(* Logix 5000 project; controller Sucrose_Main Emulate 5570 rev 20.12; software revision 20.01; part 5 of 30 *)
(* tags used below, declared in another part *)
   AI_E23_0 : REAL[8];   // Analog Input EN2T_FLX 192.168.1.23
   AI_E23_1 : REAL[8];   // Analog Input EN2T_FLX 192.168.1.23
   Alarm_ACK_Master_Timer : TIMER;
   CIPRemote : Area_Program;
   DI_E20_0 : ALIAS FOR FLX_E20:0:I;   // Discrete Input EN2T_FLX 192.168.1.20
   DI_E20_1 : ALIAS FOR FLX_E20:1:I;   // Discrete Input EN2T_FLX 192.168.1.20
   DO_E20_4 : ALIAS FOR FLX_E20:4:O;   // Discrete Output EN2T_FLX 192.168.1.20
   DO_E20_5 : ALIAS FOR FLX_E20:5:O;   // Discrete Output EN2T_FLX 192.168.1.20
   FV610501_AOI : QSI_Flow_Valve;   // FV-61-05-01-O CIP SUPPLY TO FILTRATION AND RING MAIN MIX PROOF VALVE OPEN
   FV620101_AOI : QSI_Flow_Valve;   // FV-62-01-01-O SUCROSE TANK #1 TO CIP RETURN PUMP MIX PROOF VALVE OPEN
   FV620201_AOI : QSI_Flow_Valve;   // FV-62-02-01-O SUCROSE TANK #2 TO CIP RETURN PUMP MIX PROOF VALVE OPEN
   Sucrose_MM_Enable : BOOL;
   SucroseCIP_PAUSED : BOOL;
   SucroseCIP_RINGMAIN_REMOTE : CIP_REMOTE;
   SucroseCIP_RUNNING : BOOL;
   SucroseCIP_SeatLift_Pulsing : BOOL;
   SucroseCIP_TK230101_REMOTE : CIP_REMOTE;
   SucroseCIP_TK230201_REMOTE : CIP_REMOTE;
   SucroseCIP_TK230301_REMOTE : CIP_REMOTE;
(* CIP_RemoteArea_AutoLogic, continued *)

ROUTINE CIP_TK230201_Remote   (* ladder *)
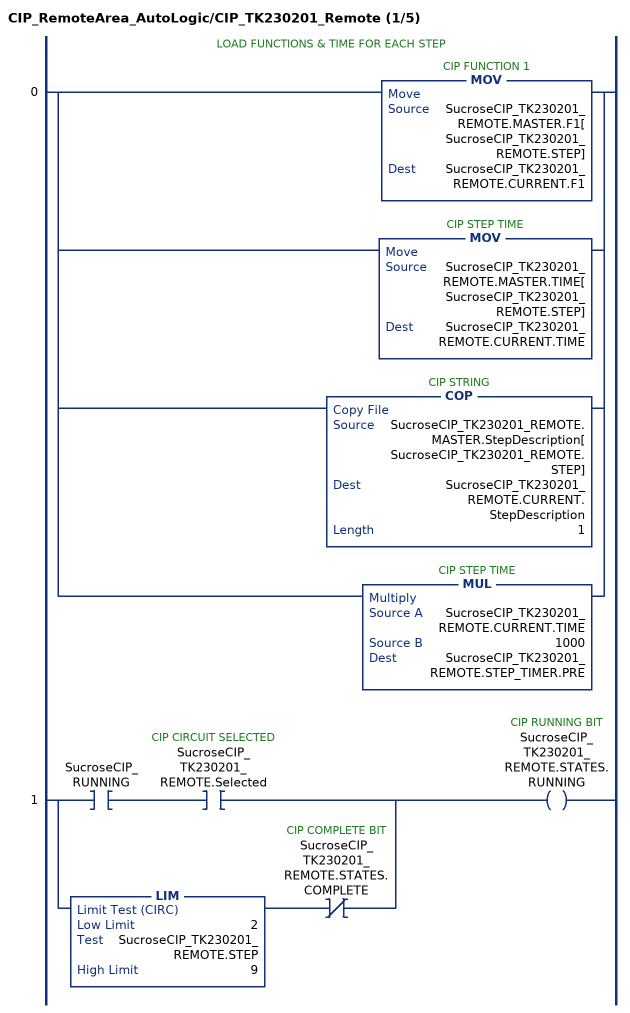
   // LOAD FUNCTIONS & TIME FOR EACH STEP
   0: [MOV(SucroseCIP_TK230201_REMOTE.MASTER.F1[SucroseCIP_TK230201_REMOTE.STEP],SucroseCIP_TK230201_REMOTE.CURRENT.F1) ,MOV(SucroseCIP_TK230201_REMOTE.MASTER.TIME[SucroseCIP_TK230201_REMOTE.STEP],SucroseCIP_TK230201_REMOTE.CURRENT.TIME) ,COP(SucroseCIP_TK230201_REMOTE.MASTER.StepDescription[SucroseCIP_TK230201_REMOTE.STEP],SucroseCIP_TK230201_REMOTE.CURRENT.StepDescription,1) ,MUL(SucroseCIP_TK230201_REMOTE.CURRENT.TIME,1000,SucroseCIP_TK230201_REMOTE.STEP_TIMER.PRE) ];
   1: [XIC(SucroseCIP_RUNNING) XIC(SucroseCIP_TK230201_REMOTE.Selected) ,LIM(2,SucroseCIP_TK230201_REMOTE.STEP,9) XIO(SucroseCIP_TK230201_REMOTE.STATES.COMPLETE) ]OTE(SucroseCIP_TK230201_REMOTE.STATES.RUNNING);
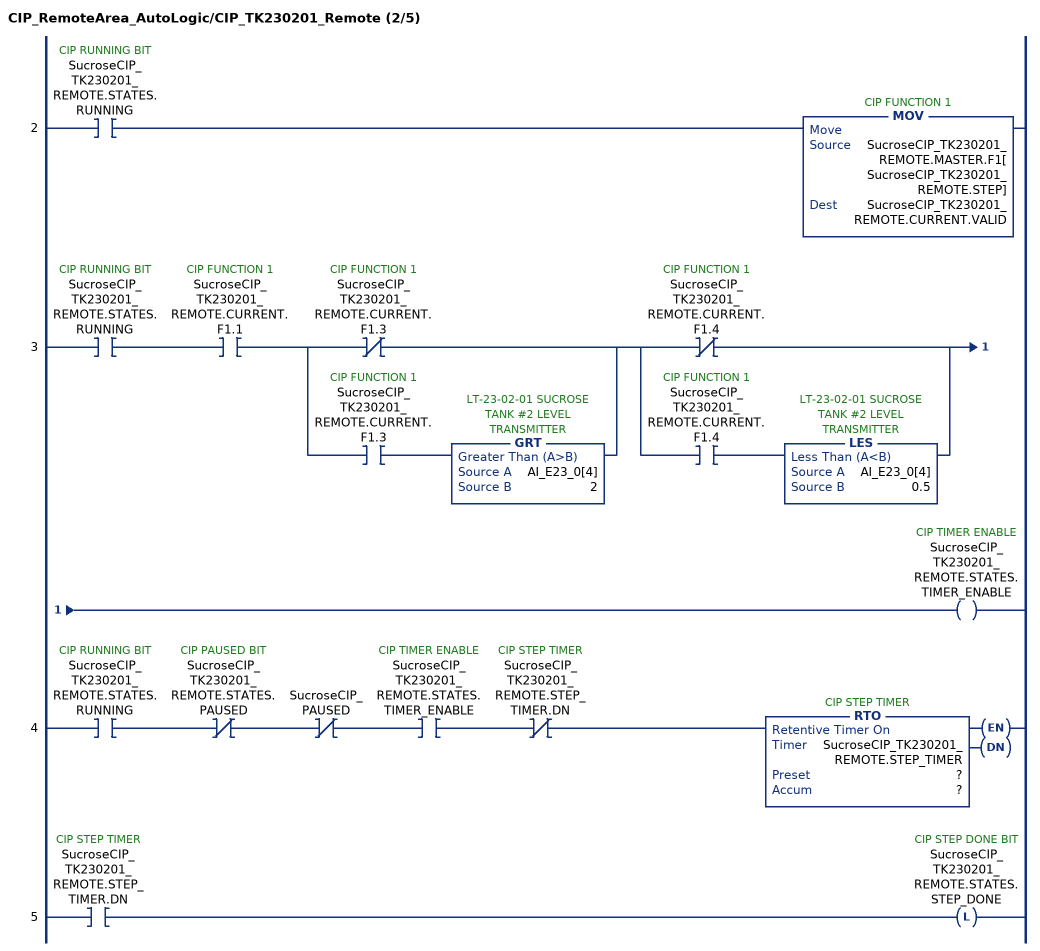
   2: XIC(SucroseCIP_TK230201_REMOTE.STATES.RUNNING)MOV(SucroseCIP_TK230201_REMOTE.MASTER.F1[SucroseCIP_TK230201_REMOTE.STEP],SucroseCIP_TK230201_REMOTE.CURRENT.VALID);
   3: XIC(SucroseCIP_TK230201_REMOTE.STATES.RUNNING)XIC(SucroseCIP_TK230201_REMOTE.CURRENT.F1.1)[XIO(SucroseCIP_TK230201_REMOTE.CURRENT.F1.3) ,XIC(SucroseCIP_TK230201_REMOTE.CURRENT.F1.3) GRT(AI_E23_0[4],2) ][XIO(SucroseCIP_TK230201_REMOTE.CURRENT.F1.4) ,XIC(SucroseCIP_TK230201_REMOTE.CURRENT.F1.4) LES(AI_E23_0[4],0.5) ]OTE(SucroseCIP_TK230201_REMOTE.STATES.TIMER_ENABLE);
   4: XIC(SucroseCIP_TK230201_REMOTE.STATES.RUNNING)XIO(SucroseCIP_TK230201_REMOTE.STATES.PAUSED)XIO(SucroseCIP_PAUSED)XIC(SucroseCIP_TK230201_REMOTE.STATES.TIMER_ENABLE)XIO(SucroseCIP_TK230201_REMOTE.STEP_TIMER.DN)RTO(SucroseCIP_TK230201_REMOTE.STEP_TIMER,?,?);
   5: XIC(SucroseCIP_TK230201_REMOTE.STEP_TIMER.DN)OTL(SucroseCIP_TK230201_REMOTE.STATES.STEP_DONE);
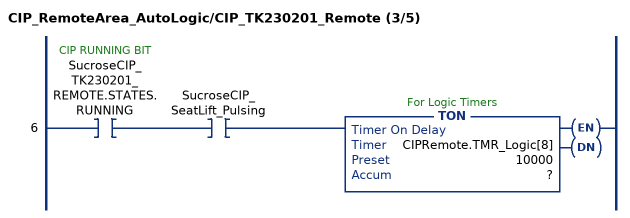
   6: XIC(SucroseCIP_TK230201_REMOTE.STATES.RUNNING)XIC(SucroseCIP_SeatLift_Pulsing)TON(CIPRemote.TMR_Logic[8],?,?);
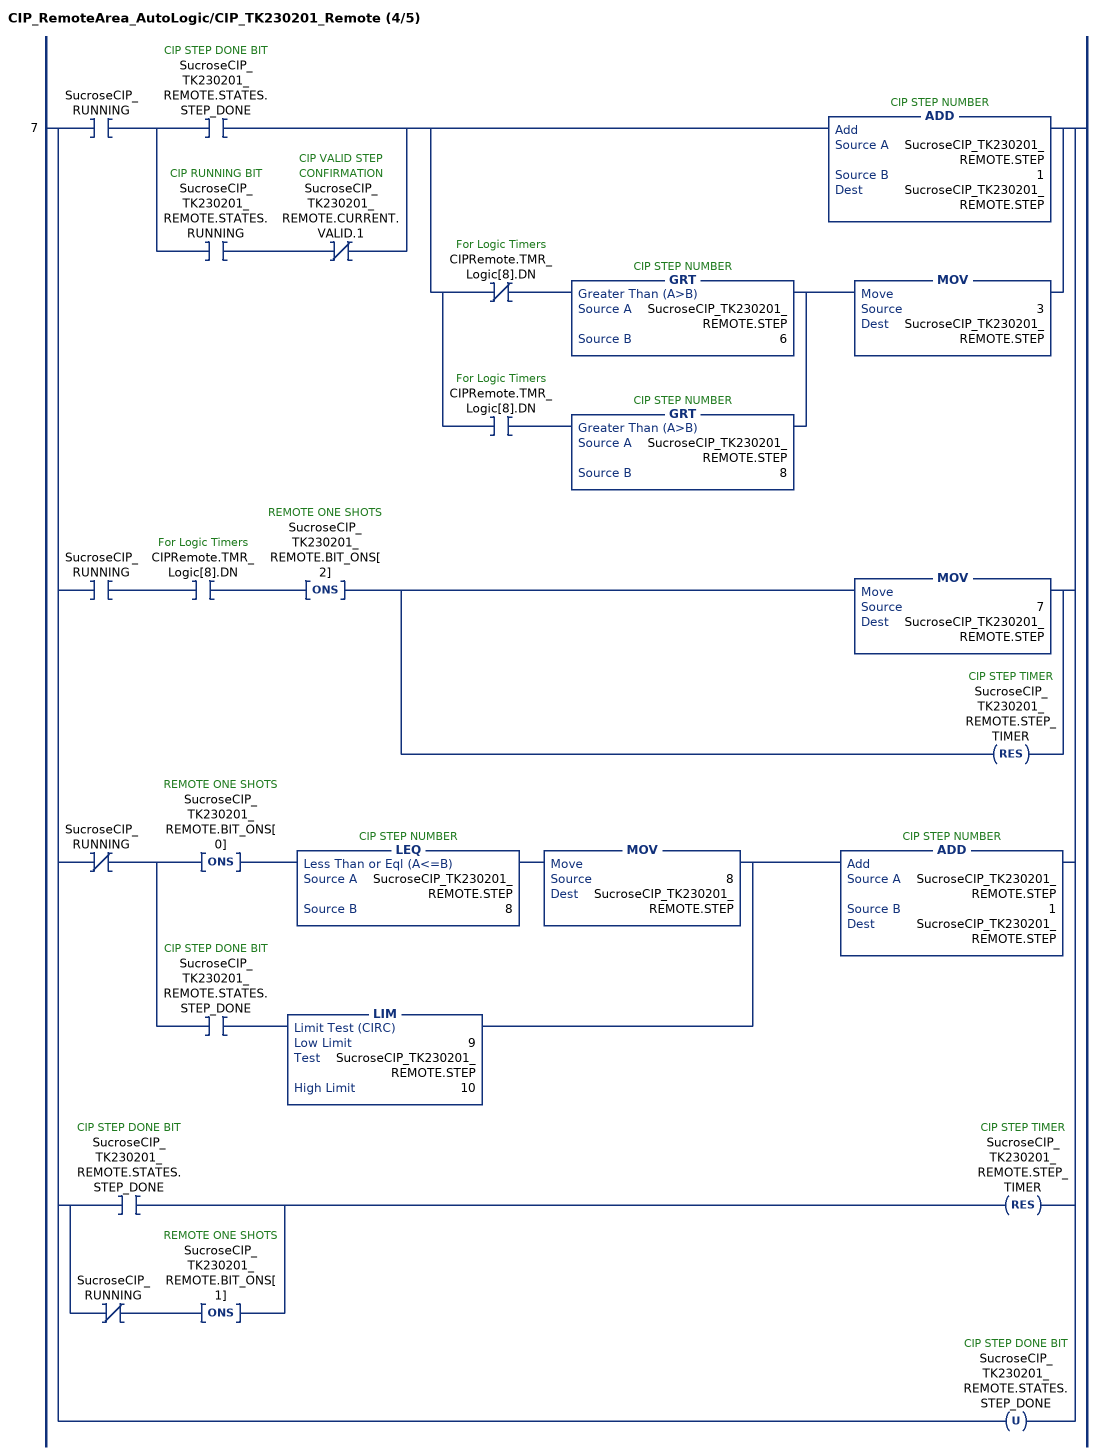
   7: [XIC(SucroseCIP_RUNNING) [XIC(SucroseCIP_TK230201_REMOTE.STATES.STEP_DONE) ,XIC(SucroseCIP_TK230201_REMOTE.STATES.RUNNING) XIO(SucroseCIP_TK230201_REMOTE.CURRENT.VALID.1) ] [ADD(SucroseCIP_TK230201_REMOTE.STEP,1,SucroseCIP_TK230201_REMOTE.STEP) ,[XIO(CIPRemote.TMR_Logic[8].DN) GRT(SucroseCIP_TK230201_REMOTE.STEP,6) ,XIC(CIPRemote.TMR_Logic[8].DN) GRT(SucroseCIP_TK230201_REMOTE.STEP,8) ] MOV(3,SucroseCIP_TK230201_REMOTE.STEP) ] ,XIC(SucroseCIP_RUNNING) XIC(CIPRemote.TMR_Logic[8].DN) ONS(SucroseCIP_TK230201_REMOTE.BIT_ONS[2]) [MOV(7,SucroseCIP_TK230201_REMOTE.STEP) ,RES(SucroseCIP_TK230201_REMOTE.STEP_TIMER) ] ,XIO(SucroseCIP_RUNNING) [ONS(SucroseCIP_TK230201_REMOTE.BIT_ONS[0]) LEQ(SucroseCIP_TK230201_REMOTE.STEP,8) MOV(8,SucroseCIP_TK230201_REMOTE.STEP) ,XIC(SucroseCIP_TK230201_REMOTE.STATES.STEP_DONE) LIM(9,SucroseCIP_TK230201_REMOTE.STEP,10) ] ADD(SucroseCIP_TK230201_REMOTE.STEP,1,SucroseCIP_TK230201_REMOTE.STEP) ,[XIC(SucroseCIP_TK230201_REMOTE.STATES.STEP_DONE) ,XIO(SucroseCIP_RUNNING) ONS(SucroseCIP_TK230201_REMOTE.BIT_ONS[1]) ] RES(SucroseCIP_TK230201_REMOTE.STEP_TIMER) ,OTU(SucroseCIP_TK230201_REMOTE.STATES.STEP_DONE) ];
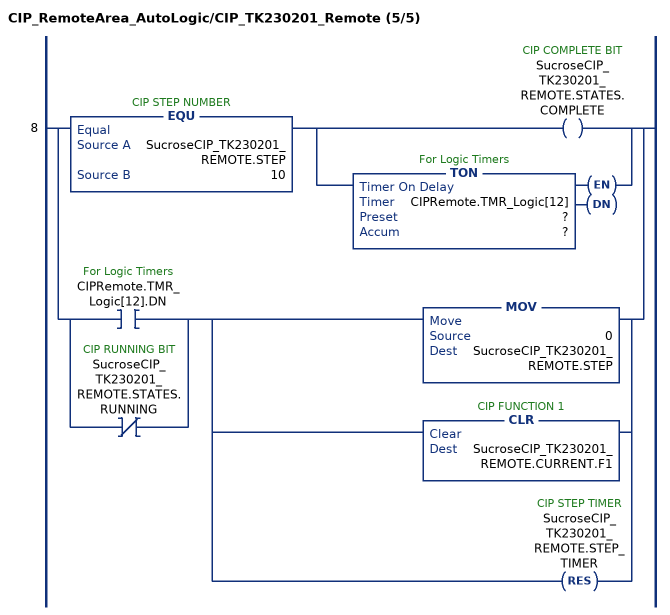
   8: [EQU(SucroseCIP_TK230201_REMOTE.STEP,10) [OTE(SucroseCIP_TK230201_REMOTE.STATES.COMPLETE) ,TON(CIPRemote.TMR_Logic[12],?,?) ] ,[XIC(CIPRemote.TMR_Logic[12].DN) ,XIO(SucroseCIP_TK230201_REMOTE.STATES.RUNNING) ] [MOV(0,SucroseCIP_TK230201_REMOTE.STEP) ,CLR(SucroseCIP_TK230201_REMOTE.CURRENT.F1) ,RES(SucroseCIP_TK230201_REMOTE.STEP_TIMER) ] ];
END_ROUTINE

ROUTINE CIP_TK230301_Remote   (* ladder *)
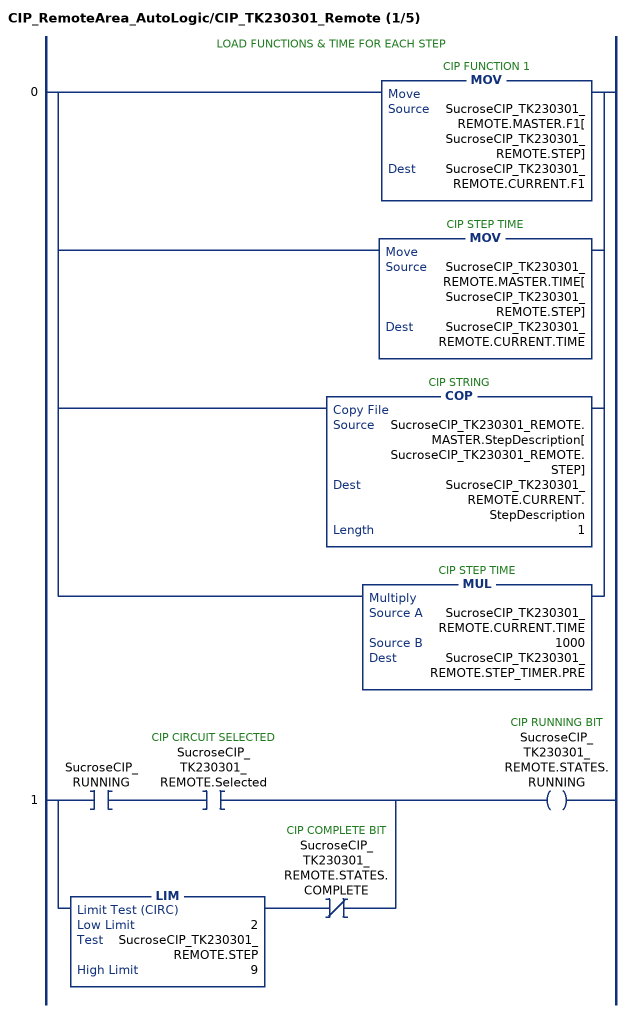
   // LOAD FUNCTIONS & TIME FOR EACH STEP
   0: [MOV(SucroseCIP_TK230301_REMOTE.MASTER.F1[SucroseCIP_TK230301_REMOTE.STEP],SucroseCIP_TK230301_REMOTE.CURRENT.F1) ,MOV(SucroseCIP_TK230301_REMOTE.MASTER.TIME[SucroseCIP_TK230301_REMOTE.STEP],SucroseCIP_TK230301_REMOTE.CURRENT.TIME) ,COP(SucroseCIP_TK230301_REMOTE.MASTER.StepDescription[SucroseCIP_TK230301_REMOTE.STEP],SucroseCIP_TK230301_REMOTE.CURRENT.StepDescription,1) ,MUL(SucroseCIP_TK230301_REMOTE.CURRENT.TIME,1000,SucroseCIP_TK230301_REMOTE.STEP_TIMER.PRE) ];
   1: [XIC(SucroseCIP_RUNNING) XIC(SucroseCIP_TK230301_REMOTE.Selected) ,LIM(2,SucroseCIP_TK230301_REMOTE.STEP,9) XIO(SucroseCIP_TK230301_REMOTE.STATES.COMPLETE) ]OTE(SucroseCIP_TK230301_REMOTE.STATES.RUNNING);
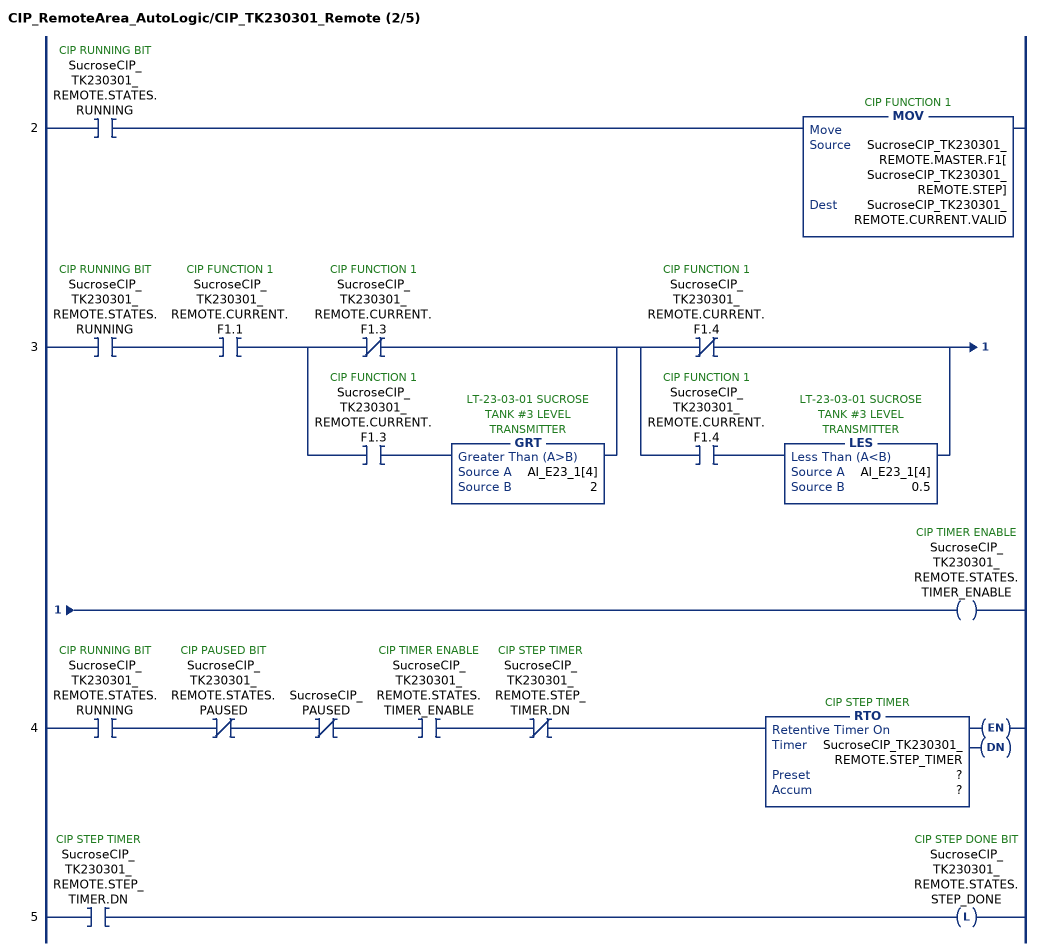
   2: XIC(SucroseCIP_TK230301_REMOTE.STATES.RUNNING)MOV(SucroseCIP_TK230301_REMOTE.MASTER.F1[SucroseCIP_TK230301_REMOTE.STEP],SucroseCIP_TK230301_REMOTE.CURRENT.VALID);
   3: XIC(SucroseCIP_TK230301_REMOTE.STATES.RUNNING)XIC(SucroseCIP_TK230301_REMOTE.CURRENT.F1.1)[XIO(SucroseCIP_TK230301_REMOTE.CURRENT.F1.3) ,XIC(SucroseCIP_TK230301_REMOTE.CURRENT.F1.3) GRT(AI_E23_1[4],2) ][XIO(SucroseCIP_TK230301_REMOTE.CURRENT.F1.4) ,XIC(SucroseCIP_TK230301_REMOTE.CURRENT.F1.4) LES(AI_E23_1[4],0.5) ]OTE(SucroseCIP_TK230301_REMOTE.STATES.TIMER_ENABLE);
   4: XIC(SucroseCIP_TK230301_REMOTE.STATES.RUNNING)XIO(SucroseCIP_TK230301_REMOTE.STATES.PAUSED)XIO(SucroseCIP_PAUSED)XIC(SucroseCIP_TK230301_REMOTE.STATES.TIMER_ENABLE)XIO(SucroseCIP_TK230301_REMOTE.STEP_TIMER.DN)RTO(SucroseCIP_TK230301_REMOTE.STEP_TIMER,?,?);
   5: XIC(SucroseCIP_TK230301_REMOTE.STEP_TIMER.DN)OTL(SucroseCIP_TK230301_REMOTE.STATES.STEP_DONE);
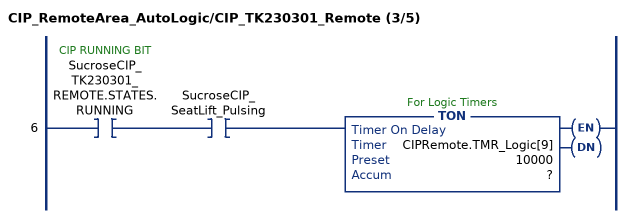
   6: XIC(SucroseCIP_TK230301_REMOTE.STATES.RUNNING)XIC(SucroseCIP_SeatLift_Pulsing)TON(CIPRemote.TMR_Logic[9],?,?);
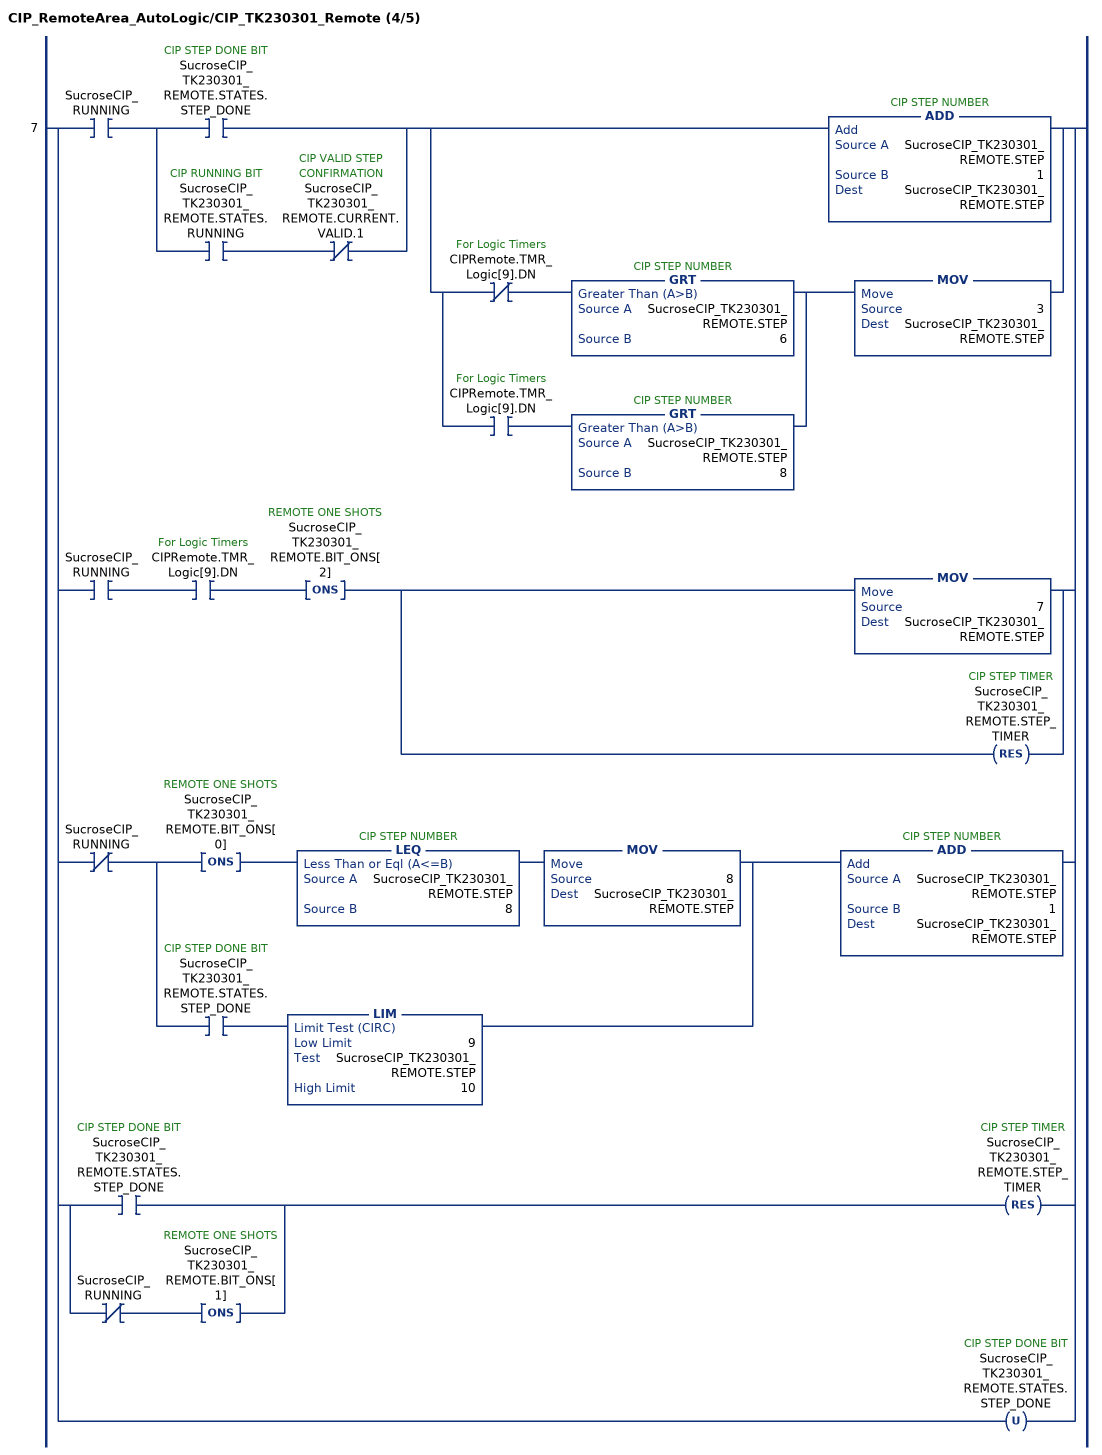
   7: [XIC(SucroseCIP_RUNNING) [XIC(SucroseCIP_TK230301_REMOTE.STATES.STEP_DONE) ,XIC(SucroseCIP_TK230301_REMOTE.STATES.RUNNING) XIO(SucroseCIP_TK230301_REMOTE.CURRENT.VALID.1) ] [ADD(SucroseCIP_TK230301_REMOTE.STEP,1,SucroseCIP_TK230301_REMOTE.STEP) ,[XIO(CIPRemote.TMR_Logic[9].DN) GRT(SucroseCIP_TK230301_REMOTE.STEP,6) ,XIC(CIPRemote.TMR_Logic[9].DN) GRT(SucroseCIP_TK230301_REMOTE.STEP,8) ] MOV(3,SucroseCIP_TK230301_REMOTE.STEP) ] ,XIC(SucroseCIP_RUNNING) XIC(CIPRemote.TMR_Logic[9].DN) ONS(SucroseCIP_TK230301_REMOTE.BIT_ONS[2]) [MOV(7,SucroseCIP_TK230301_REMOTE.STEP) ,RES(SucroseCIP_TK230301_REMOTE.STEP_TIMER) ] ,XIO(SucroseCIP_RUNNING) [ONS(SucroseCIP_TK230301_REMOTE.BIT_ONS[0]) LEQ(SucroseCIP_TK230301_REMOTE.STEP,8) MOV(8,SucroseCIP_TK230301_REMOTE.STEP) ,XIC(SucroseCIP_TK230301_REMOTE.STATES.STEP_DONE) LIM(9,SucroseCIP_TK230301_REMOTE.STEP,10) ] ADD(SucroseCIP_TK230301_REMOTE.STEP,1,SucroseCIP_TK230301_REMOTE.STEP) ,[XIC(SucroseCIP_TK230301_REMOTE.STATES.STEP_DONE) ,XIO(SucroseCIP_RUNNING) ONS(SucroseCIP_TK230301_REMOTE.BIT_ONS[1]) ] RES(SucroseCIP_TK230301_REMOTE.STEP_TIMER) ,OTU(SucroseCIP_TK230301_REMOTE.STATES.STEP_DONE) ];
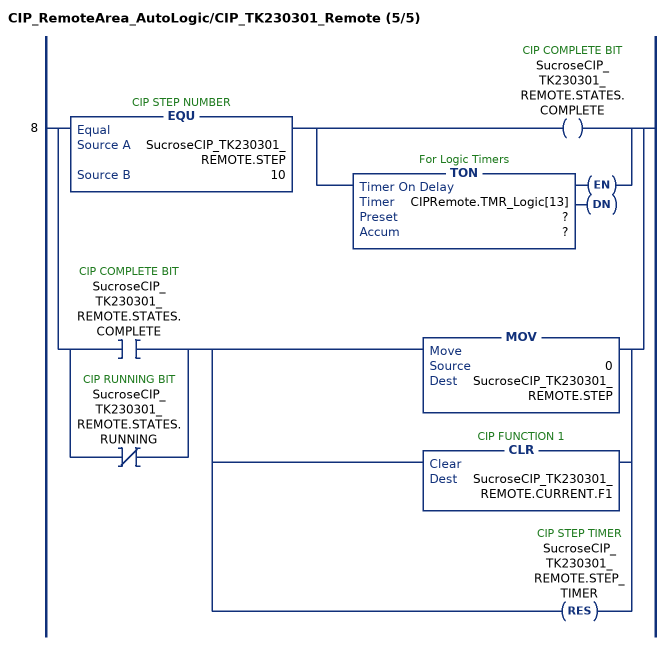
   8: [EQU(SucroseCIP_TK230301_REMOTE.STEP,10) [OTE(SucroseCIP_TK230301_REMOTE.STATES.COMPLETE) ,TON(CIPRemote.TMR_Logic[13],?,?) ] ,[XIC(SucroseCIP_TK230301_REMOTE.STATES.COMPLETE) ,XIO(SucroseCIP_TK230301_REMOTE.STATES.RUNNING) ] [MOV(0,SucroseCIP_TK230301_REMOTE.STEP) ,CLR(SucroseCIP_TK230301_REMOTE.CURRENT.F1) ,RES(SucroseCIP_TK230301_REMOTE.STEP_TIMER) ] ];
END_ROUTINE

ROUTINE MainRoutine   (* ladder *)
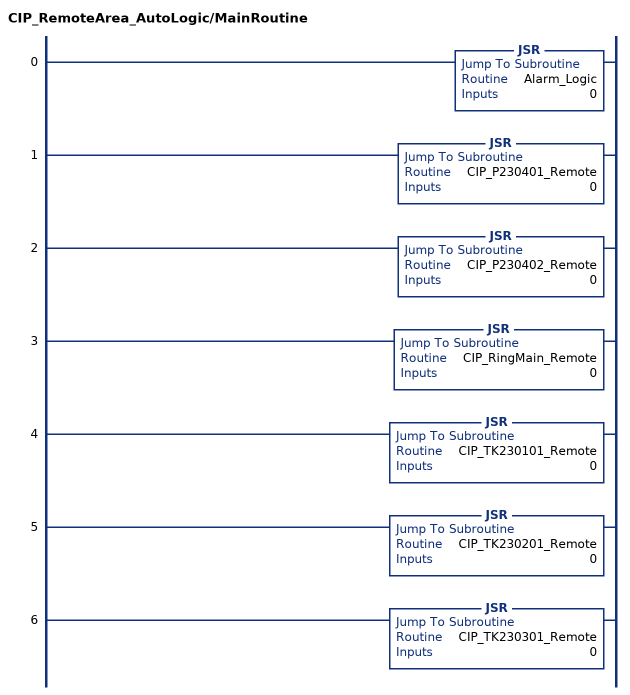
   0: JSR(Alarm_Logic,0);
   1: JSR(CIP_P230401_Remote,0);
   2: JSR(CIP_P230402_Remote,0);
   3: JSR(CIP_RingMain_Remote,0);
   4: JSR(CIP_TK230101_Remote,0);
   5: JSR(CIP_TK230201_Remote,0);
   6: JSR(CIP_TK230301_Remote,0);
END_ROUTINE
END_PROGRAM

PROGRAM CIP_RemoteArea_EN2T_IO_Discrete_DO_E20_4   (* main routine MainRoutine *)

ROUTINE _00_FV610501   (* ladder *)
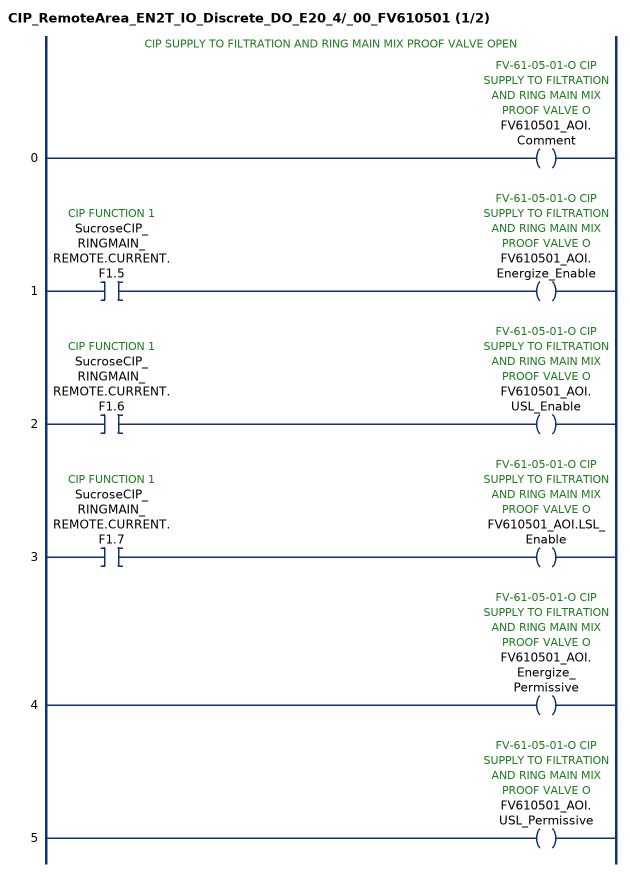
   // CIP SUPPLY TO FILTRATION AND RING MAIN MIX PROOF VALVE OPEN
   0: OTE(FV610501_AOI.Comment);
   1: XIC(SucroseCIP_RINGMAIN_REMOTE.CURRENT.F1.5)OTE(FV610501_AOI.Energize_Enable);
   2: XIC(SucroseCIP_RINGMAIN_REMOTE.CURRENT.F1.6)OTE(FV610501_AOI.USL_Enable);
   3: XIC(SucroseCIP_RINGMAIN_REMOTE.CURRENT.F1.7)OTE(FV610501_AOI.LSL_Enable);
   4: OTE(FV610501_AOI.Energize_Permissive);
   5: OTE(FV610501_AOI.USL_Permissive);
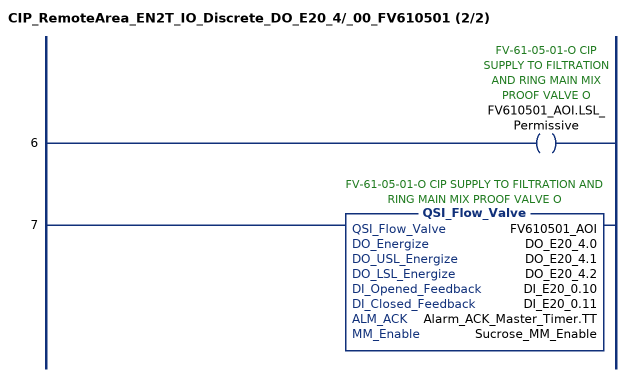
   6: OTE(FV610501_AOI.LSL_Permissive);
   7: QSI_Flow_Valve(FV610501_AOI,DO_E20_4.0,DO_E20_4.1,DO_E20_4.2,DI_E20_0.10,DI_E20_0.11,Alarm_ACK_Master_Timer.TT,Sucrose_MM_Enable);
END_ROUTINE

ROUTINE _12_FV620101   (* ladder *)
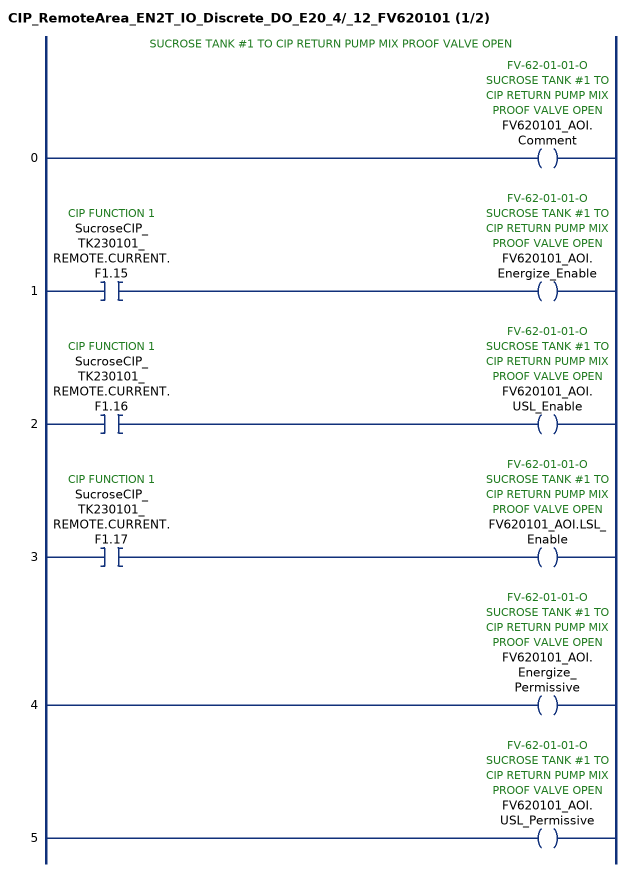
   // SUCROSE TANK #1 TO CIP RETURN PUMP MIX PROOF VALVE OPEN
   0: OTE(FV620101_AOI.Comment);
   1: XIC(SucroseCIP_TK230101_REMOTE.CURRENT.F1.15)OTE(FV620101_AOI.Energize_Enable);
   2: XIC(SucroseCIP_TK230101_REMOTE.CURRENT.F1.16)OTE(FV620101_AOI.USL_Enable);
   3: XIC(SucroseCIP_TK230101_REMOTE.CURRENT.F1.17)OTE(FV620101_AOI.LSL_Enable);
   4: OTE(FV620101_AOI.Energize_Permissive);
   5: OTE(FV620101_AOI.USL_Permissive);
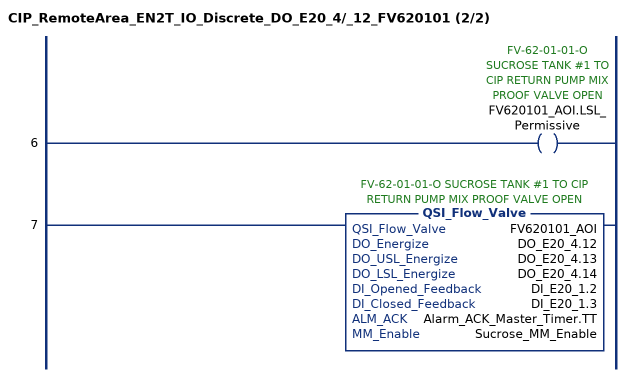
   6: OTE(FV620101_AOI.LSL_Permissive);
   7: QSI_Flow_Valve(FV620101_AOI,DO_E20_4.12,DO_E20_4.13,DO_E20_4.14,DI_E20_1.2,DI_E20_1.3,Alarm_ACK_Master_Timer.TT,Sucrose_MM_Enable);
END_ROUTINE

ROUTINE MainRoutine   (* ladder *)
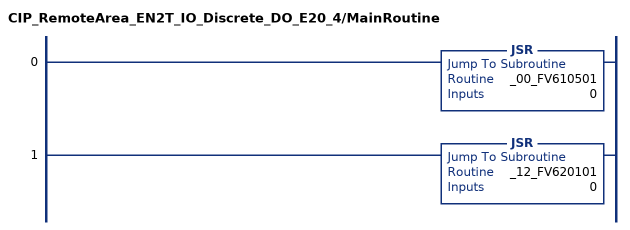
   0: JSR(_00_FV610501,0);
   1: JSR(_12_FV620101,0);
END_ROUTINE
END_PROGRAM

PROGRAM CIP_RemoteArea_EN2T_IO_Discrete_DO_E20_5   (* main routine MainRoutine *)

ROUTINE _00_FV620201   (* ladder *)
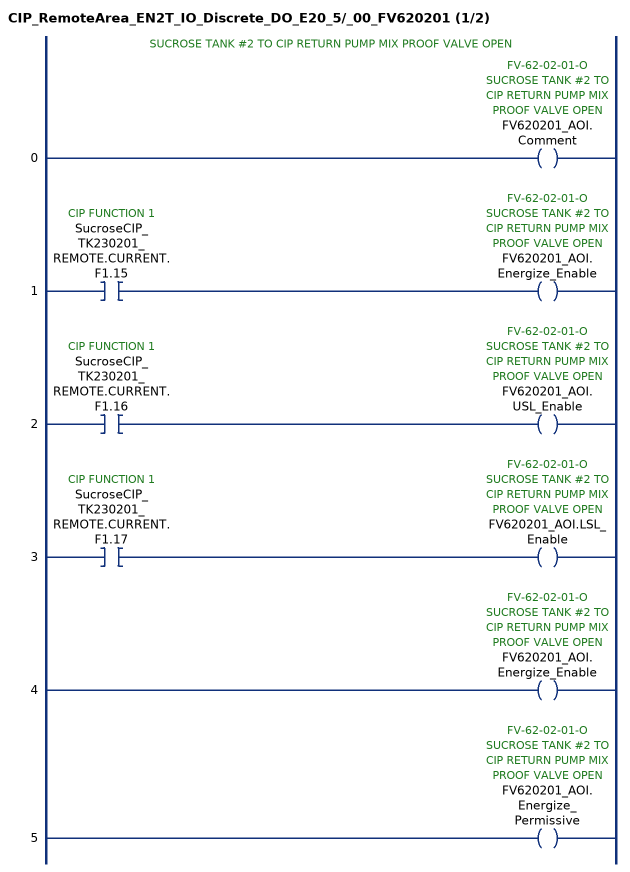
   // SUCROSE TANK #2 TO CIP RETURN PUMP MIX PROOF VALVE OPEN
   0: OTE(FV620201_AOI.Comment);
   1: XIC(SucroseCIP_TK230201_REMOTE.CURRENT.F1.15)OTE(FV620201_AOI.Energize_Enable);
   2: XIC(SucroseCIP_TK230201_REMOTE.CURRENT.F1.16)OTE(FV620201_AOI.USL_Enable);
   3: XIC(SucroseCIP_TK230201_REMOTE.CURRENT.F1.17)OTE(FV620201_AOI.LSL_Enable);
   4: OTE(FV620201_AOI.Energize_Enable);
   5: OTE(FV620201_AOI.Energize_Permissive);
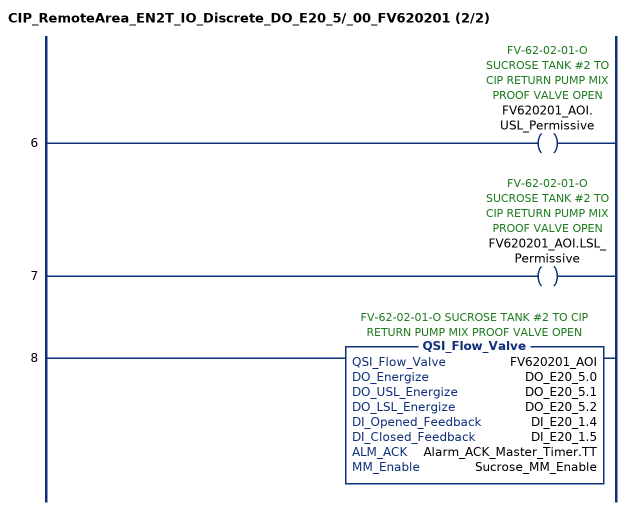
   6: OTE(FV620201_AOI.USL_Permissive);
   7: OTE(FV620201_AOI.LSL_Permissive);
   8: QSI_Flow_Valve(FV620201_AOI,DO_E20_5.0,DO_E20_5.1,DO_E20_5.2,DI_E20_1.4,DI_E20_1.5,Alarm_ACK_Master_Timer.TT,Sucrose_MM_Enable);
END_ROUTINE
